Fanuc KAREL source: kt00092.KL

-- PROVISIONAL review KL for V1013-1; original PC SHA256 7ec9915b6de414d925aad998eeb54ced6545c62c4eacc98e10d39c39ed382793
-- Incomplete behavior may be omitted. Consult companion uncertainty JSON. Do not deploy.
PROGRAM KT00092
%NOLOCKGROUP
VAR
  R2 : REAL
  OUT : REAL
-- UNRESOLVED_DECL H1 type=002017
BEGIN
  -- UNRESOLVED_PC offsets 5-19; opcodes 2E,22,9D,33,B4
  -- UNRESOLVED_PC offsets 24-35; opcodes 2E,23
  -- UNRESOLVED_PC offsets 40-64; opcodes 22,9D,33,B3,21,29,64,6B,23
  -- UNRESOLVED_PC offsets 69-73; opcodes 7F
END KT00092
